FUNCTION_BLOCK FB_FastThreadConfig
VAR
END_VAR

METHOD FB_Exit : BOOL
VAR_INPUT
	bInCopyCode: BOOL;
END_VAR
IF NOT bInCopyCode THEN
	GVL_OnlineChangeTest.StageState.iConfiguredFastThread := 0;
	GVL_OnlineChangeTest.StageState.bFastThreadConfigured := FALSE;
END_IF
END_METHOD

METHOD FB_Init : BOOL
VAR_INPUT
	bInitRetains: BOOL;
	bInCopyCode: BOOL;
	iThread: Stage.I_Thread;
END_VAR
GVL_OnlineChangeTest.StageState.iConfiguredFastThread := iThread;
END_METHOD

END_FUNCTION_BLOCK

(* stored: Version 1.1.0.1
   POU FB_FastThreadConfig: Id {42ff1aeb-9055-432c-af33-219bca3358fa}, SpecialFunc None
   Method FB_Exit: Id {3d238f9a-d8d9-4ce6-99a8-237d21dab466}
   Method FB_Init: Id {c532530f-adac-48a9-ae5e-5573e50b648f} *)
